// TIA Portal V17 export
// export: Created 2023-04-03T06:31:26.6551912Z, ExportSetting WithDefaults, DisplayName Totally Integrated Automation Portal, DisplayVersion V17 Update 4, DisplayName TIA Portal Openness, DisplayVersion V17 Update 4, DisplayName TIA Portal Version Control Interface, DisplayVersion V17, DisplayName STEP 7 Professional, DisplayVersion V17 Update 4, DisplayName STEP 7 Safety, DisplayVersion V17, DisplayName WinCC Professional, DisplayVersion V17 Update 4
FUNCTION "PCS W (F)_1" : Void   // FC48, LAD
TITLE = ModBus TCP for PCS Power Electronics
{ S7_Optimized_Access := 'TRUE' }
VERSION : 0.1
// stored: AutoNumber true, IsIECCheckEnabled false, SetENOAutomatically false, UDAEnableTagReadback false
   VAR_TEMP
      rSS1PacRef : Real;
      rSS2PacRef : Real;
      rSS1QacRef : Real;
      rSS2QacRef : Real;
      rSnHalfPE : Real;
      rQacRef : Real;
      uiQacRef : UInt;
   END_VAR
   VAR_TEMP   // added for the SCL form of the ladder/FBD networks
      _w1 : Bool;
   END_VAR
BEGIN

REGION Network 1: Function Modbus Client
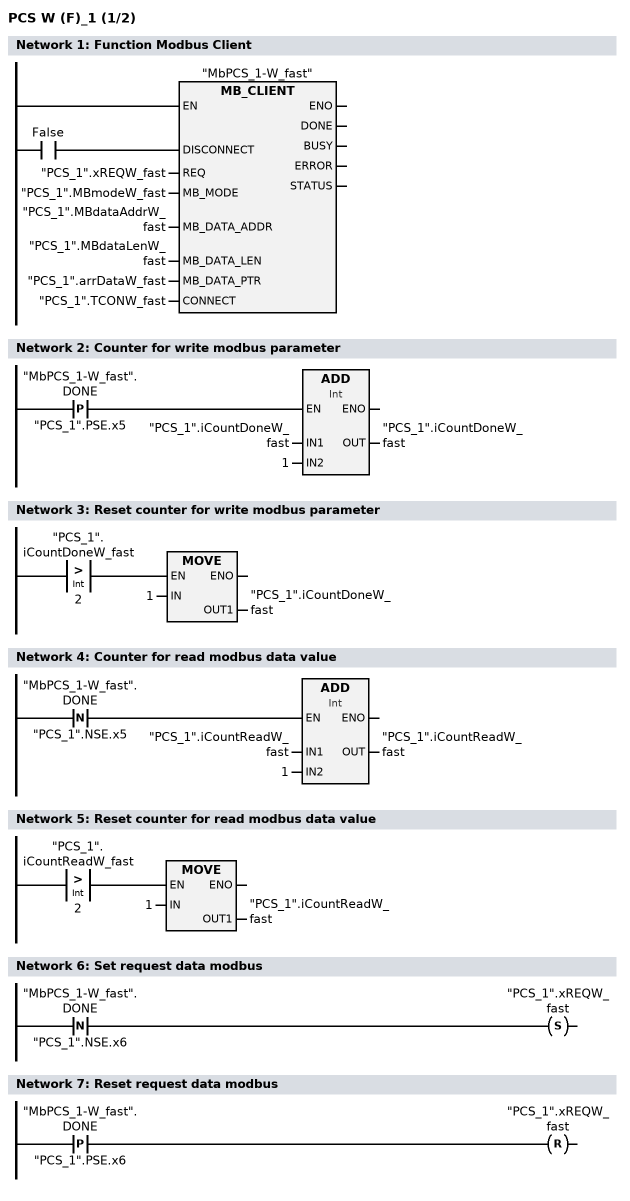
   RUNG wire#powerrail
      "MbPCS_1-W_fast".MB_CLIENT(DISCONNECT := wire#w1, REQ := "PCS_1".xREQW_fast, MB_MODE := "PCS_1".MBmodeW_fast, MB_DATA_ADDR := "PCS_1".MBdataAddrW_fast, MB_DATA_LEN := "PCS_1".MBdataLenW_fast, MB_DATA_PTR := "PCS_1".arrDataW_fast, CONNECT := "PCS_1".TCONW_fast, DONE =>, BUSY =>, ERROR =>, STATUS =>)
   END_RUNG
   RUNG wire#powerrail
      Contact( False )
   END_RUNG wire#w1
   // the same network as SCL:
   "MbPCS_1-W_fast"(DISCONNECT := False,   // MB_CLIENT
                    REQ := "PCS_1".xREQW_fast,
                    MB_MODE := "PCS_1".MBmodeW_fast,
                    MB_DATA_ADDR := "PCS_1".MBdataAddrW_fast,
                    MB_DATA_LEN := "PCS_1".MBdataLenW_fast,
                    MB_DATA_PTR := "PCS_1".arrDataW_fast,
                    CONNECT := "PCS_1".TCONW_fast);
END_REGION

REGION Network 2: Counter for write modbus parameter
   RUNG wire#powerrail
      P_Contact(operand := "MbPCS_1-W_fast".DONE, bit := "PCS_1".PSE.x5)
      { S7_Templates := "SrcType := Int" } Add(in1 := "PCS_1".iCountDoneW_fast, in2 := 1, out => "PCS_1".iCountDoneW_fast)
   END_RUNG
   // the same network as SCL:
   #_w1 := "MbPCS_1-W_fast".DONE AND NOT "PCS_1".PSE.x5;   // rising edge of "MbPCS_1-W_fast".DONE
   "PCS_1".PSE.x5 := "MbPCS_1-W_fast".DONE;
   IF #_w1 THEN "PCS_1".iCountDoneW_fast := "PCS_1".iCountDoneW_fast + 1; END_IF;
END_REGION

REGION Network 3: Reset counter for write modbus parameter
   RUNG wire#powerrail
      { S7_Templates := "SrcType := Int" } GT_Contact(in1 := "PCS_1".iCountDoneW_fast, in2 := 2)
      Move(in := 1, out1 => "PCS_1".iCountDoneW_fast)
   END_RUNG
   // the same network as SCL:
   IF "PCS_1".iCountDoneW_fast > 2 THEN "PCS_1".iCountDoneW_fast := 1; END_IF;
END_REGION

REGION Network 4: Counter for read modbus data value
   RUNG wire#powerrail
      N_Contact(operand := "MbPCS_1-W_fast".DONE, bit := "PCS_1".NSE.x5)
      { S7_Templates := "SrcType := Int" } Add(in1 := "PCS_1".iCountReadW_fast, in2 := 1, out => "PCS_1".iCountReadW_fast)
   END_RUNG
   // the same network as SCL:
   #_w1 := NOT "MbPCS_1-W_fast".DONE AND "PCS_1".NSE.x5;   // falling edge of "MbPCS_1-W_fast".DONE
   "PCS_1".NSE.x5 := "MbPCS_1-W_fast".DONE;
   IF #_w1 THEN "PCS_1".iCountReadW_fast := "PCS_1".iCountReadW_fast + 1; END_IF;
END_REGION

REGION Network 5: Reset counter for read modbus data value
   RUNG wire#powerrail
      { S7_Templates := "SrcType := Int" } GT_Contact(in1 := "PCS_1".iCountReadW_fast, in2 := 2)
      Move(in := 1, out1 => "PCS_1".iCountReadW_fast)
   END_RUNG
   // the same network as SCL:
   IF "PCS_1".iCountReadW_fast > 2 THEN "PCS_1".iCountReadW_fast := 1; END_IF;
END_REGION

REGION Network 6: Set request data modbus
   RUNG wire#powerrail
      N_Contact(operand := "MbPCS_1-W_fast".DONE, bit := "PCS_1".NSE.x6)
      S_Coil( "PCS_1".xREQW_fast )
   END_RUNG
   // the same network as SCL:
   #_w1 := NOT "MbPCS_1-W_fast".DONE AND "PCS_1".NSE.x6;   // falling edge of "MbPCS_1-W_fast".DONE
   "PCS_1".NSE.x6 := "MbPCS_1-W_fast".DONE;
   IF #_w1 THEN "PCS_1".xREQW_fast := TRUE; END_IF;
END_REGION

REGION Network 7: Reset request data modbus
   RUNG wire#powerrail
      P_Contact(operand := "MbPCS_1-W_fast".DONE, bit := "PCS_1".PSE.x6)
      R_Coil( "PCS_1".xREQW_fast )
   END_RUNG
   // the same network as SCL:
   #_w1 := "MbPCS_1-W_fast".DONE AND NOT "PCS_1".PSE.x6;   // rising edge of "MbPCS_1-W_fast".DONE
   "PCS_1".PSE.x6 := "MbPCS_1-W_fast".DONE;
   IF #_w1 THEN "PCS_1".xREQW_fast := FALSE; END_IF;
END_REGION

REGION Network 9: Write Active Power Reference
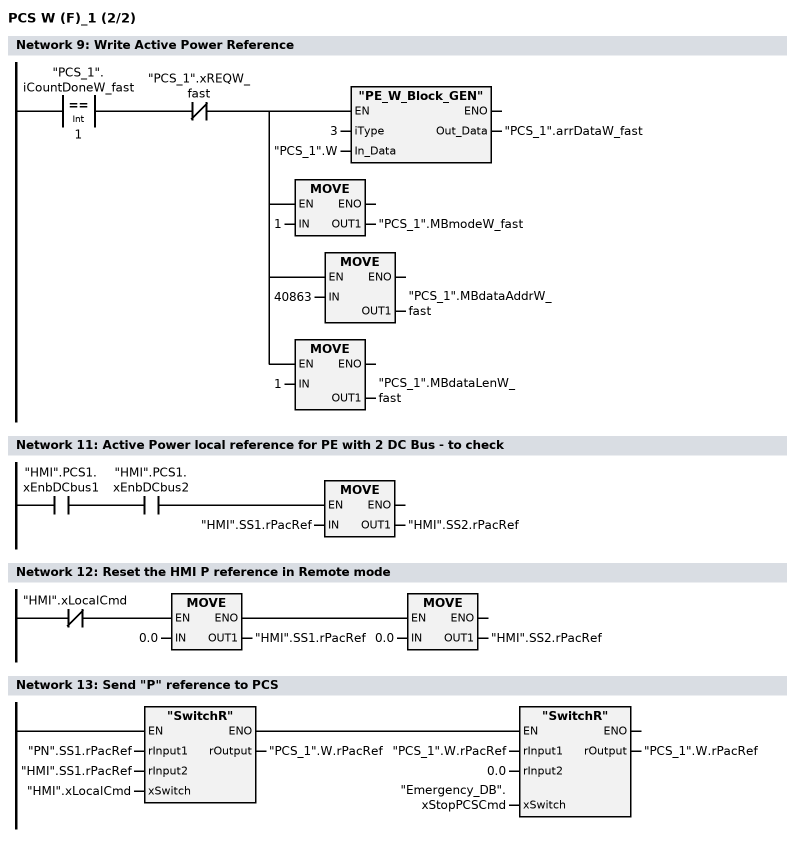
   RUNG wire#powerrail
      { S7_Templates := "SrcType := Int" } EQ_Contact(in1 := "PCS_1".iCountDoneW_fast, in2 := 1)
      I_Contact( "PCS_1".xREQW_fast )
      wire#w1
      "PE_W_Block_GEN"(iType := 3, In_Data := "PCS_1".W, Out_Data => "PCS_1".arrDataW_fast)
   END_RUNG
   RUNG wire#w1
      Move(in := 1, out1 => "PCS_1".MBmodeW_fast)
   END_RUNG
   RUNG wire#w1
      Move(in := 40863, out1 => "PCS_1".MBdataAddrW_fast)
   END_RUNG
   RUNG wire#w1
      Move(in := 1, out1 => "PCS_1".MBdataLenW_fast)
   END_RUNG
   // the same network as SCL:
   #_w1 := ("PCS_1".iCountDoneW_fast = 1) AND NOT "PCS_1".xREQW_fast;
   IF #_w1 THEN
       "PE_W_Block_GEN"(iType := 3, In_Data := "PCS_1".W, Out_Data => "PCS_1".arrDataW_fast);
       "PCS_1".MBmodeW_fast := 1;
       "PCS_1".MBdataAddrW_fast := 40863;
       "PCS_1".MBdataLenW_fast := 1;
   END_IF;
END_REGION

REGION Network 11: Active Power local reference for PE with 2 DC Bus - to check
   RUNG wire#powerrail
      Contact( "HMI".PCS1.xEnbDCbus1 )
      Contact( "HMI".PCS1.xEnbDCbus2 )
      Move(in := "HMI".SS1.rPacRef, out1 => "HMI".SS2.rPacRef)
   END_RUNG
   // the same network as SCL:
   IF "HMI".PCS1.xEnbDCbus1 AND "HMI".PCS1.xEnbDCbus2 THEN "HMI".SS2.rPacRef := "HMI".SS1.rPacRef; END_IF;
END_REGION

REGION Network 12: Reset the HMI P reference in Remote mode
   RUNG wire#powerrail
      I_Contact( "HMI".xLocalCmd )
      Move(in := 0.0, out1 => "HMI".SS1.rPacRef)
      Move(in := 0.0, out1 => "HMI".SS2.rPacRef)
   END_RUNG
   // the same network as SCL:
   IF NOT "HMI".xLocalCmd THEN
       "HMI".SS1.rPacRef := 0.0;
       "HMI".SS2.rPacRef := 0.0;
   END_IF;
END_REGION

REGION Network 13: Send "P" reference to PCS
   RUNG wire#powerrail
      "SwitchR"(rInput1 := "PN".SS1.rPacRef, rInput2 := "HMI".SS1.rPacRef, xSwitch := "HMI".xLocalCmd, rOutput => "PCS_1".W.rPacRef)
      "SwitchR"(rInput1 := "PCS_1".W.rPacRef, rInput2 := 0.0, xSwitch := "Emergency_DB".xStopPCSCmd, rOutput => "PCS_1".W.rPacRef)
   END_RUNG
   // the same network as SCL:
   "SwitchR"(rInput1 := "PN".SS1.rPacRef,
             rInput2 := "HMI".SS1.rPacRef,
             xSwitch := "HMI".xLocalCmd,
             rOutput => "PCS_1".W.rPacRef,
             ENO => #_w1);
   IF #_w1 THEN
       "SwitchR"(rInput1 := "PCS_1".W.rPacRef,
                 rInput2 := 0.0,
                 xSwitch := "Emergency_DB".xStopPCSCmd,
                 rOutput => "PCS_1".W.rPacRef);
   END_IF;
END_REGION
END_FUNCTION
